Staubli VAL3: OnF1.pgx

program OnF1()
  local bool l_bRes
begin

  pPoint[sItem]=here(flange,world)

end
